{attribute 'qualified_only'}
{attribute 'strict'}
TYPE eFBERROR :
(   
	(*Function block errors*)
	NoError								:=0,
	WrongFilePath						:=101,
	WrongDS6_ProcessPath				:=103,
	WrongEtherCATRevision				:=105,
	InvalidBoxname						:=107,
	WrongServiceTypeInput				:=109,
	TimeoutExceed						:=111,
	NoStoberSlaveInConfiguration		:=113,
	
	(*DS6 Errors*)
	ProjectNotFound						:=201,//Drive controller project not found
	MoreThanOneProjectFound				:=203,//Drive Controller found several times in project 
	OpenProjectError					:=205,//project open error 
	ConnectionError						:=207,//Connection to Drive controller failed 
	OnlineError							:=209//Online connection failed 
	
	


);
END_TYPE

(* stored: Version 1.1.0.1, ProductVersion 3.1.4024.6
   EnumerationTextList eFBERROR: Id {f1f614b5-a32b-40a2-9438-41e32fa4c5d6} *)
